Universal Robots PolyScope program: Operation.urp

Program Operation (createdIn=3.5.1.10661 lastSavedIn=3.5.1.10661 directory=/programs/usbdisk installation=default robotSerialNumber=2018333842)
Calibrated DH parameters: a=[0.000044, -0.212779, -0.212115, 0.000007, -0.000103, 0]; d=[0.152199, 116.652206, -129.176863, 12.637137, 0.085345, 0.08253]; alpha=[1.570557, -0.001022, -0.001933, 1.570765, -1.571025, 0]; deltaTheta=[0.000019, -0.511005, 0.624572, -0.11359, -0.000034, 0.000065]
BeforeStart
  freeze_move := False
  var_1 := socket_open("192.168.88.13",30000)
  targetPos := [0,0,0,0,0,0]
  prevPos := [0,0,0,0,0,0]
  delay := 0
  counter := 0
  flag := 0
  grip := 0
  MoveJ speed 60 deg/s, acceleration 80 deg/s^2 (useActiveTCP=false)
    Waypoint base_pos: TCP in base x=329.969 y=-101.94 z=328.457 mm, rx=3.0559 ry=0.0782 rz=0.0831 rad; joints [3, -95, -82, -90, 85, 270] deg
Robot Program (runOnlyOnce=false motionType=MoveJ speed=1.047198 acceleration=1.396263 useActiveTCP=false)
  Loop While (checkContinuously=false) expression=var_1≟ False
    var_1 := socket_open("192.168.88.13",30000)
  Script: socket_send_string("sensor_val")
  var_2 := socket_read_ascii_float(8)
  If var_2[0]≟8
    If var_2[7]≟1
      grip := 0
    Else 
      grip := 1
    delay := var_2[8]
    Loop While (checkContinuously=false) expression=counter<6
      Script: targetPos[counter] = var_2[counter+1]
      counter := counter+1
    flag := 0
  var_1 := False
  Script: socket_close()
  counter := 0
  flag := 1
Thread Thread_2 (runOnlyOnce=false trackProgramExecution=false)
  If grip≟1
    URCap Gripper (Robotiq_Grippers, Robotiq Inc.) dataModel(position=100.0, force=100.0, speed=100.0, positionInDouble=100.0, forceInDouble=100.0, speedInDouble=100.0, slaveIds=[9], blocking=true); state(isChildrenLocked=true)
  Else 
    URCap Gripper (Robotiq_Grippers, Robotiq Inc.) dataModel(position=0.0, force=100.0, speed=100.0, positionInDouble=0.0, forceInDouble=100.0, speedInDouble=100.0, slaveIds=[9], blocking=true); state(isChildrenLocked=true)
Thread Thread_1 (runOnlyOnce=false trackProgramExecution=false)
  If flag≟1 (checkContinuously=true)
    If targetPos≠prevPos  and  targetPos≠[0,0,0,0,0,0]
      Script: movej(targetPos,a=1.4,v=1.5,t=delay,r=0)
      Script: prevPos=targetPos
  Else 
    Script: stopj(15)
  Wait Sleep waitTime=0.001
